//VALVES
// Pump Isolation Valves
// FB_VRC
//EBD Side
//TURBO
fb_AT1K0_GAS_VRC_10(i_xExtILK_OK := F_TurboGateValve_ILK(fb_AT1K0_GAS_PTM_10.iq_stPtm,fb_AT1K0_GAS_GPI_10.PG), i_xOverrideMode := xSystemOverrideMode);
fb_AT1K0_GAS_VRC_20(i_xExtILK_OK := F_TurboGateValve_ILK(fb_AT1K0_GAS_PTM_20.iq_stPtm,fb_AT1K0_GAS_GPI_20.PG), i_xOverrideMode := xSystemOverrideMode);
fb_AT1K0_GAS_VRC_30(i_xExtILK_OK := F_TurboGateValve_ILK(fb_AT1K0_GAS_PTM_30.iq_stPtm,fb_AT1K0_GAS_GPI_30.PG), i_xOverrideMode := xSystemOverrideMode);
fb_AT1K0_GAS_VRC_40(i_xExtILK_OK := F_TurboGateValve_ILK(fb_AT1K0_GAS_PTM_40.iq_stPtm,fb_AT1K0_GAS_GPI_40.PG), i_xOverrideMode := xSystemOverrideMode);
//EBD
fb_AT1K0_GAS_VRC_50(i_xExtILK_OK := F_VRC_DIODE_ILK(fb_AT1K0_GAS_GPI_50.PG,fb_AT1K0_GAS_GPI_51.PG), i_xOverrideMode := xSystemOverrideMode);
fb_AT1K0_GAS_VRC_60(i_xExtILK_OK := F_VRC_DIODE_ILK(fb_AT1K0_GAS_GPI_60.PG,fb_AT1K0_GAS_GPI_51.PG), i_xOverrideMode := xSystemOverrideMode);
//FEE Side
fb_AT1K0_GAS_VRC_70(i_xExtILK_OK := fb_AT1K0_GAS_PMF_90.stPump.i_xMPStatus, i_xOverrideMode := xSystemOverrideMode);
fb_AT1K0_GAS_VRC_90(i_xExtILK_OK := fb_AT1K0_GAS_PMF_90.stPump.i_xMPStatus, i_xOverrideMode := xSystemOverrideMode);
fb_AT1K0_GAS_VRC_100(i_xExtILK_OK := fb_AT1K0_GAS_PMF_100.stPump.i_xMPStatus, i_xOverrideMode := xSystemOverrideMode);
//TURBO
fb_AT1K0_GAS_VRC_110(i_xExtILK_OK := F_TurboGateValve_ILK(fb_AT1K0_GAS_PTM_110.iq_stPtm,fb_AT1K0_GAS_GPI_110.PG), i_xOverrideMode := xSystemOverrideMode);
fb_AT1K0_GAS_VRC_120(i_xExtILK_OK := F_TurboGateValve_ILK(fb_AT1K0_GAS_PTM_120.iq_stPtm,fb_AT1K0_GAS_GPI_120.PG), i_xOverrideMode := xSystemOverrideMode);
fb_AT1K0_GAS_VRC_130(i_xExtILK_OK := F_TurboGateValve_ILK(fb_AT1K0_GAS_PTM_130.iq_stPtm,fb_AT1K0_GAS_GPI_130.PG), i_xOverrideMode := xSystemOverrideMode);
fb_AT1K0_GAS_VRC_140(i_xExtILK_OK := F_TurboGateValve_ILK(fb_AT1K0_GAS_PTM_140.iq_stPtm,fb_AT1K0_GAS_GPI_140.PG) , i_xOverrideMode := xSystemOverrideMode);
//N2 valve
//INL VCN, VGP and VRC_70 are closed.
fb_AT1K0_GAS_VRC_80.i_xExtILK_OK := fb_AT1K0_GAS_VRC_90.iq_stValve.i_xClsLS AND VCN_70.iq_stVCN.rReqPosition <0.4 AND VVC_71.M_IsClosed() AND VVC_72.M_IsClosed() ; //AND VGP is closed;
fb_AT1K0_GAS_VRC_80( i_xOverrideMode := xSystemOverrideMode);


// Turbo Pumps
// FB_PTM_Ebara_010M
//EBD SIDE
fb_AT1K0_GAS_PTM_10(i_xExtILKOk := F_TurboExtILKLogic_2(fb_AT1K0_GAS_PTM_10.iq_stPtm, fb_AT1K0_GAS_GPI_11.PG, fb_AT1K0_GAS_GPI_10.PG,fb_AT1K0_GAS_PMF_10.iq_stPFO));
fb_AT1K0_GAS_PTM_20(i_xExtILKOk := F_TurboExtILKLogic_2(fb_AT1K0_GAS_PTM_20.iq_stPtm, fb_AT1K0_GAS_GPI_11.PG, fb_AT1K0_GAS_GPI_20.PG,fb_AT1K0_GAS_PMF_10.iq_stPFO));
fb_AT1K0_GAS_PTM_30(i_xExtILKOk := F_TurboExtILKLogic_2(fb_AT1K0_GAS_PTM_30.iq_stPtm, fb_AT1K0_GAS_GPI_11.PG, fb_AT1K0_GAS_GPI_30.PG,fb_AT1K0_GAS_PMF_10.iq_stPFO));
fb_AT1K0_GAS_PTM_40(i_xExtILKOk := F_TurboExtILKLogic_2(fb_AT1K0_GAS_PTM_40.iq_stPtm, fb_AT1K0_GAS_GPI_11.PG, fb_AT1K0_GAS_GPI_40.PG,fb_AT1K0_GAS_PMF_10.iq_stPFO));
//FEE Side
fb_AT1K0_GAS_PTM_110(i_xExtILKOk := F_TurboExtILKLogic_2(fb_AT1K0_GAS_PTM_110.iq_stPtm, fb_AT1K0_GAS_GPI_111.PG,fb_AT1K0_GAS_GPI_110.PG,fb_AT1K0_GAS_PMF_110.stPump));
fb_AT1K0_GAS_PTM_120(i_xExtILKOk := F_TurboExtILKLogic_2(fb_AT1K0_GAS_PTM_120.iq_stPtm, fb_AT1K0_GAS_GPI_121.PG, fb_AT1K0_GAS_GPI_120.PG,fb_AT1K0_GAS_PMF_120.stPump));
fb_AT1K0_GAS_PTM_130(i_xExtILKOk := F_TurboExtILKLogic_2(fb_AT1K0_GAS_PTM_130.iq_stPtm, fb_AT1K0_GAS_GPI_121.PG,fb_AT1K0_GAS_GPI_130.PG,fb_AT1K0_GAS_PMF_120.stPump)); 
fb_AT1K0_GAS_PTM_140(i_xExtILKOk := F_TurboExtILKLogic_2(fb_AT1K0_GAS_PTM_140.iq_stPtm, fb_AT1K0_GAS_GPI_141.PG,fb_AT1K0_GAS_GPI_140.PG,fb_AT1K0_GAS_PMF_140.stPump));

// Injector side
fb_AT1K0_GAS_VVC_80(i_xExtILK_OK:= (fb_AT1K0_GAS_PMF_110.stPump.eState = pumpRUNNING  OR  fb_AT1K0_GAS_PMF_110.stPump.eState = pumpSTARTING ) AND (fb_AT1K0_GAS_PTM_80.iq_stPtm.eState = pumpSTARTING OR fb_AT1K0_GAS_PTM_80.iq_stPtm.eState = pumpRUNNING) , i_xOverrideMode:= xSystemOverrideMode , iq_stValve=> );
fb_AT1K0_GAS_PTM_80(i_xExtILKOk := F_TurboExtILKLogic_2(fb_AT1K0_GAS_PTM_80.iq_stPtm, fb_AT1K0_GAS_GPI_111.PG,fb_AT1K0_GAS_GPI_80.PG,fb_AT1K0_GAS_PMF_110.stPump));

//Rouging pumps
// FB_EbaraDryPump
//EBD SIDE
fb_AT1K0_GAS_PMF_10(xExtIlk :=TRUE,TurboIsOn := TRUE);
fb_AT1K0_GAS_PMF_60(xExtIlk :=TRUE,TurboIsOn := TRUE);
//FEE SIDE
fb_AT1K0_GAS_PMF_90(i_stBPGauge := fb_AT1K0_GAS_GPI_90.PG, i_xVlvOpn := TRUE, i_xExtIlkOK := TRUE);
fb_AT1K0_GAS_PMF_100(i_stBPGauge := fb_AT1K0_GAS_GPI_100.PG, i_xVlvOpn := TRUE, i_xExtIlkOK := TRUE);
fb_AT1K0_GAS_PMF_110(i_xExtIlkOK:= TRUE (*Interlock Timer on the Rough Valve*) , stPump=> );
fb_AT1K0_GAS_PMF_120(i_xExtIlkOK:= TRUE(*Interlock Timer on the Rough Valve*), stPump=> );
fb_AT1K0_GAS_PMF_140(i_xExtIlkOK:= TRUE(*Interlock Timer on the Rough Valve*), stPump=> );
if( fb_AT1K0_GAS_PMF_110.stPump.eState = pumpSTARTING ) OR ( fb_AT1K0_GAS_PMF_110.stPump.eState = pumpRUNNING ) THEN fb_AT1K0_GAS_VVC_110.M_Open(TRUE); END_IF
if( fb_AT1K0_GAS_PMF_120.stPump.eState = pumpSTARTING ) OR ( fb_AT1K0_GAS_PMF_120.stPump.eState = pumpRUNNING ) THEN fb_AT1K0_GAS_VVC_120.M_Open(TRUE); END_IF
if( fb_AT1K0_GAS_PMF_140.stPump.eState = pumpSTARTING ) OR ( fb_AT1K0_GAS_PMF_140.stPump.eState = pumpRUNNING ) THEN fb_AT1K0_GAS_VVC_140.M_Open(TRUE); END_IF
fb_AT1K0_GAS_VVC_110(i_xExtILK_OK:= (fb_AT1K0_GAS_PMF_110.stPump.eState = pumpRUNNING  OR  fb_AT1K0_GAS_PMF_110.stPump.eState = pumpSTARTING ), i_xOverrideMode:= , iq_stValve=> );
fb_AT1K0_GAS_VVC_120(i_xExtILK_OK:= (fb_AT1K0_GAS_PMF_120.stPump.eState = pumpRUNNING  OR  fb_AT1K0_GAS_PMF_120.stPump.eState = pumpSTARTING ), i_xOverrideMode:= , iq_stValve=> );
fb_AT1K0_GAS_VVC_140(i_xExtILK_OK:= (fb_AT1K0_GAS_PMF_140.stPump.eState = pumpRUNNING  OR  fb_AT1K0_GAS_PMF_140.stPump.eState = pumpSTARTING ), i_xOverrideMode:= , iq_stValve=> );

END_PROGRAM

// ---- POUs/PRG_INJ.TcPOU
PROGRAM PRG_INJ
VAR
	{attribute 'pytmc' :=' pv: AT1K0:GATT:CNTRL:SP '}
	fSetpointValue :FLOAT; 
	{attribute 'pytmc' :=' pv: AT1K0:GATT:CNTRL:GO;
	 field: ZNAM STOP; 
	 field: ONAM START; 
	 io: io;
	'}
	bGo: BOOL; 
 	{attribute 'pytmc' :=' pv: AT1K0:GATT:CNTRL:RESET;
	 field: ZNAM FALSE; 
	 field: ONAM TRUE; 
	 io: io;
	 '}
	bReset : BOOL; 
	{attribute 'pytmc' :=' pv: AT1K0:GATT:CNTRL:ERROR;
    field: ZNAM FALSE; 
	 field: ONAM TRUE; 
	 io: io;
	 '}
	bError : BOOL; 
	{attribute 'pytmc' :=' pv: AT1K0:GATT:CNTRL:Kp1 '}
	fKp1 : REAL:= 0.04; 
	{attribute 'pytmc' :=' pv: AT1K0:GATT:CNTRL:Tn1 '}
	fTn1 : REAL:= 1;//0.5; 
	{attribute 'pytmc' :=' pv: AT1K0:GATT:CNTRL:Kp2 '}
	fKp2 : REAL:= 0.01; 
	{attribute 'pytmc' :=' pv: AT1K0:GATT:CNTRL:Tn2 '}
	fTn2 : REAL:= 0.5; 
	arrTable	: ARRAY[1..31,1..2] OF FLOAT;
	fManValue											: FLOAT;
	bExtrapolate										: BOOL;
	eMode							: E_CTRL_MODE;
	stCTRL_PID_PARAMS		: ST_CTRL_PID_PARAMS;
	bSync							: BOOL;
	bHold							: BOOL;
	eErrorId						: E_CTRL_ERRORCODES;
	bARWactive					: BOOL;
	(* controller *)
	fbCTRL_PID					: FB_CTRL_PID;
	bInit							: BOOL	:= TRUE;
	fbCTRL_LIN_INTERPOLATION					: FB_CTRL_LIN_INTERPOLATION;
	//stCTRL_LIN_INTERPOLATION_PARAMS		: ST_CTRL_LIN_INTERPOLATION_PARAMS;
	stCTRL_LIN_INTERPOLATION_PARAMS_GEM	: ST_CTRL_LIN_INTERPOLATION_PARAMS;
	fbCTRL_DEADBAND						: FB_CTRL_DEADBAND;
	stCTRL_DEADBAND_PARAMS			: ST_CTRL_DEADBAND_PARAMS;

	pid_on :TON;
	wait : time := T#10S;
	FTrig: F_TRIG;
		

	
END_VAR


// Valves
VCN_70(i_xExtIlkOK := ((US_MAA_OK AND US_Roughing_Valves_Open AND US_Turbo_Valves_Open AND US_Turbo_Running) 
						AND (DS_MAA_OK AND DS_Roughing_Valves_Open AND DS_Turbo_Valves_Open AND DS_Turbo_Running)), 
						i_ReqPos:=  fbCTRL_LIN_INTERPOLATION.fOut + fbCTRL_PID.fOut);

//VGP_80
VVC_71(i_xExtILK_OK:= VVC_72.M_IsClosed(), i_xOverrideMode:= , iq_stValve=> );
VVC_72(i_xExtILK_OK:= VVC_71.M_IsClosed(), i_xOverrideMode:= , iq_stValve=> );

//Gauges
GCM_70(PG=> , i_rFULL_SCALE:= 2000);
GCM_80(PG=> , i_rFULL_SCALE:= 20);
GCM_81(PG=> , i_rFULL_SCALE:= 0.25);
(*Assign reading to psuedo gauge*)
IF (GCM_81.PG.rPRESS >=0.22) THEN GCM_82 := GCM_80.PG;
	ELSE
	GCM_82 := GCM_81.PG;	
END_IF
// Set ADC bits for EL3174-0002
GCM_70.M_SetBits(30518);
GCM_80.M_SetBits(30518);
GCM_81.M_SetBits(30518);


//
(*Iniitialization*)
IF bInit
THEN
	(* init array with the interpolation points  *)
	(* 	fIn					 |		fOut		*)
	arrTable[1,1] := 0;		arrTable[1,2] := 0;
	arrTable[2,1] := 0.0000412;		arrTable[2,2] := 34;
	arrTable[3,1] := 0.001282;		arrTable[3,2] := 36;
	arrTable[4,1] :=  0.002136;	    arrTable[4,2] := 38;
	arrTable[5,1] :=  0.005884;	    arrTable[5,2] := 40;
	arrTable[6,1] := 0.00907;		arrTable[6,2] := 42;
	arrTable[7,1] := 0.01183;		arrTable[7,2] := 44;
	arrTable[8,1] := 0.01799;	    arrTable[8,2] := 46;
	arrTable[9,1] := 0.0302;	    arrTable[9,2] := 47;
	arrTable[10,1] := 0.0417;		arrTable[10,2] := 50;
	arrTable[11,1] := 0.06635;		arrTable[11,2] := 51;
	arrTable[12,1] := 0.08118;		arrTable[12,2] := 53;
	arrTable[13,1] := 0.0998;		arrTable[13,2] := 56;
	arrTable[14,1] := 0.10644;		arrTable[14,2] := 56.5;
	arrTable[15,1] := 0.1359;		arrTable[15,2] := 58;
	arrTable[16,1] := 0.1929;		arrTable[16,2] := 60;
	arrTable[17,1] := 0.2922;		arrTable[17,2] := 62;
	arrTable[18,1] := 0.3428;	    arrTable[18,2] := 64;
	arrTable[19,1] :=  0.405;;	    arrTable[19,2] :=66;
	arrTable[20,1] := 0.481;		arrTable[20,2] := 68;
	arrTable[21,1] := 0.5542;		arrTable[21,2] := 69;
	arrTable[22,1] := 0.6333;	    arrTable[22,2] := 70;
	arrTable[23,1] := 0.7901;	    arrTable[23,2] := 72;
	arrTable[24,1] := 0.9307;		arrTable[24,2] := 73.04;
	arrTable[25,1] := 1.0448;		arrTable[25,2] := 73.64;
	arrTable[26,1] := 1.31919;;		arrTable[26,2] := 74.45;
	arrTable[27,1] :=  1.324;		arrTable[27,2] :=74.46;
	arrTable[28,1] := 1.71941;	arrTable[28,2] := 75;
	arrTable[29,1] :=  1.963194;		arrTable[29,2] :=75.5;
	arrTable[30,1] := 1.99999;	arrTable[30,2] := 75.505;
	arrTable[31,1] := 2;	arrTable[31,2] := 75.55;
	(* init parameter struct *)
	stCTRL_LIN_INTERPOLATION_PARAMS_GEM.tCtrlCycleTime					:= T#10ms;
	stCTRL_LIN_INTERPOLATION_PARAMS_GEM.tTaskCycleTime					:= T#10ms;
	stCTRL_LIN_INTERPOLATION_PARAMS_GEM.nDataTable_NumberOfRows		:= INT_TO_UINT(31);	

	(*FBCNTRL*)
	(* init parameter struct *)
	stCTRL_PID_PARAMS.tCtrlCycleTime		:= T#10ms;
	stCTRL_PID_PARAMS.tTaskCycleTime		:= T#10ms;
	stCTRL_PID_PARAMS.fKp					:= fKp1;			(* proportional gain Kp				*)
	stCTRL_PID_PARAMS.tTn					:= T#500ms;		(*  Tn									*)
	stCTRL_PID_PARAMS.tTv					:= T#200ms;	(*  Tv									*)
	stCTRL_PID_PARAMS.tTd					:= T#100ms;	(*  Td									*)
	stCTRL_PID_PARAMS.fOutMaxLimit			:=  78;			(* maximum output limit				*)
	stCTRL_PID_PARAMS.fOutMinLimit			:=  -100;			(* minimum output limit				*)

	(* set the mode to ACTIVE --> normal operation *)
	eMode							:= eCTRL_MODE_ACTIVE   ;					
	(* reset the init flag *)
	bInit							:= FALSE;
END_IF
(* set the addresses *)
	stCTRL_LIN_INTERPOLATION_PARAMS_GEM.pDataTable_ADR			:= ADR(arrTable);
	stCTRL_LIN_INTERPOLATION_PARAMS_GEM.nDataTable_SIZEOF		:= SIZEOF(arrTable);

if (bGo) THEN
	IF (bReset) THEN
	(* set the mode to RESET*)
	eMode							:= eCTRL_MODE_RESET   ;
	VCN_70.M_ValveControl(CloseValve);
	//bReset := False;
	ELSE
		(* set the mode to ACTIVE --> normal operation *)
	eMode							:= eCTRL_MODE_ACTIVE   ;
 	VCN_70.M_ValveControl(PressureControl);
	END_IF
END_IF
If(FTrig.Q)THEN
		eMode							:= eCTRL_MODE_PASSIVE;
		VCN_70.M_ValveControl(CloseValve);
		fSetpointValue :=0;
END_IF


fbCTRL_LIN_INTERPOLATION(
	fIn:= fSetpointValue , 
	fManValue:= fManValue , 
	bExtrapolate:= bExtrapolate, 
	eMode:= eMode, 
	stParams:= stCTRL_LIN_INTERPOLATION_PARAMS_GEM,
	fOut=> , 
	bInIsGreaterThanMaxElement=> , 
	bInIsLessThanMinElement=> , 
	eState=> , 
	eErrorId=> , 
	bError=> );


(* Gauge selection *)
IF (fSetpointValue >=0.22) THEN
	fbCTRL_PID.fActualValue := GCM_80.PG.rPRESS;
ELSE
	fbCTRL_PID.fActualValue := GCM_81.PG.rPRESS;
END_IF

(* call controller *)
fbCTRL_PID(		fSetpointValue		:= fSetpointValue,
					fActualValue		:= ,
					fManSyncValue	:= ,
					bSync				:= bSync,
					eMode				:= eMode,
					bHold				:= bHold,
					stParams			:= stCTRL_PID_PARAMS,
					fOut				=> ,
					bARWactive		=> bARWactive,
					eErrorId			=> eErrorId,
					bError				=> 
				);

	
(*deadband/clipper *)

(* call function block *)
stCTRL_DEADBAND_PARAMS.fThreshold	:=  fSetpointValue*0.0016 ;
(*fbCTRL_DEADBAND	(	fIn					:= ,
					stParams			:= stCTRL_DEADBAND_PARAMS,
					bInIsUnderThreshold => ,
					eErrorId			=> ,
					bError				=> 
				);*)

bError := fbCTRL_PID.bError OR fbCTRL_LIN_INTERPOLATION.bError;
				

	

// or NOT???

//stCTRL_PID_PARAMS.bDInTheFeedbackPath := fbCTRL_DEADBAND.bInIsUnderThreshold;


//timer
(*pid_on(IN:=, PT:= wait, Q=>, ET =>);
IF (pid_on.Q) THEN eMode:= eCTRL_MODE_ACTIVE; pid_on.IN := FALSE; END_IF; //eCTRL_MODE_TUNE????*)


FTRIG(CLK := bGo);

END_PROGRAM

// ---- POUs/PRG_Motion.TcPOU
PROGRAM PRG_Motion
VAR
	bInit: BOOL := TRUE;
	iReqApperture: INT :=1;
	
	bAllGo : Bool := false;
	
	/////
 (* fbMAX_1: FB_MotionStage;
  fbMAY_1: FB_MotionStage;
  
  fbMAX_2: FB_MotionStage;
  fbMAY_2: FB_MotionStage;
  
  fbMAX_3: FB_MotionStage;
  fbMAY_3: FB_MotionStage;
  
  fbMAX_4: FB_MotionStage;
  fbMAY_4: FB_MotionStage;*)
	
	/////
	{attribute 'pytmc' := '
		pv: MMS:1:STATE
		io: io
	'}
	fbMAA_1_States: FB_MAA;
	{attribute 'pytmc' := '
		pv: MMS:2:STATE
		io: io
	'}
	fbMAA_2_States: FB_MAA;
	{attribute 'pytmc' := '
		pv: MMS:3:STATE
		io: io
	'}
	fbMAA_3_States: FB_MAA;
	{attribute 'pytmc' := '
		pv: MMS:4:STATE
		io: io
	'}
	fbMAA_4_States: FB_MAA;

END_VAR

/// PMPS ???????????
//LIMIT the array index
iReqApperture := LIMIT(1,pv_iReqApperture,4);


(*
IF(bInit) THEN
	// initialise all the values of pre defined positions for each apperture in the assembly array 
	VAA_1_Y_POS[1] :=0;
	VAA_1_Y_POS[2] :=0;
	VAA_1_Y_POS[3] :=0;
	VAA_1_Y_POS[4] :=0;
	
	VAA_2_Y_POS[1] :=0;
	VAA_2_Y_POS[2] :=0;
	VAA_2_Y_POS[3] :=0;
	VAA_2_Y_POS[4] :=0;
	
	VAA_3_Y_POS[1] :=0;
	VAA_3_Y_POS[2] :=0;
	VAA_3_Y_POS[3] :=0;
	VAA_3_Y_POS[4] :=0;
	
	VAA_4_Y_POS[1] :=0;
	VAA_4_Y_POS[2] :=0;
	VAA_4_Y_POS[3] :=0;
	VAA_4_Y_POS[4] :=0;
END_IF


(*No STO*)
M1.bHardwareEnable := TRUE;
M2.bHardwareEnable := TRUE;
M3.bHardwareEnable := TRUE;
M4.bHardwareEnable := TRUE;

M5.bHardwareEnable := TRUE;
M6.bHardwareEnable := TRUE;
M7.bHardwareEnable := TRUE;
M8.bHardwareEnable := TRUE;

(*Instantiate the motion function blocks*)
fbMAX_1(stMotionStage := M1);
fbMAY_1(stMotionStage := M2);

fbMAX_2(stMotionStage := M3);
fbMAY_2(stMotionStage := M4);

fbMAX_3(stMotionStage := M4);
fbMAY_3(stMotionStage := M6);

fbMAX_4(stMotionStage := M7);
fbMAY_4(stMotionStage := M8);

(* PTP to aperture position on the each aperture array assembly*)
fbMAA_1_States(
	stMotionStage:=M2,
	fbGoAprt1:=VAA_1_Y_POS[1],
	fbGoAprt2:=VAA_1_Y_POS[2],
	fbGoAprt3:=VAA_1_Y_POS[3],
	fbGoAprt4:=VAA_1_Y_POS[4]);

fbMAA_2_States(
	stMotionStage:=M4,
	fbGoAprt1:=VAA_2_Y_POS[1],
	fbGoAprt2:=VAA_2_Y_POS[2],
	fbGoAprt3:=VAA_2_Y_POS[3],
	fbGoAprt4:=VAA_2_Y_POS[4]);
	
fbMAA_3_States(
	stMotionStage:=M6,
	fbGoAprt1:=VAA_3_Y_POS[1],
	fbGoAprt2:=VAA_3_Y_POS[2],
	fbGoAprt3:=VAA_3_Y_POS[3],
	fbGoAprt4:=VAA_3_Y_POS[4]);
	
fbMAA_4_States(
	stMotionStage:=M8,
	fbGoAprt1:=VAA_4_Y_POS[1],
	fbGoAprt2:=VAA_4_Y_POS[2],
	fbGoAprt3:=VAA_4_Y_POS[3],
	fbGoAprt4:=VAA_4_Y_POS[4]);
	
If (bAllGo) Then

	CASE iReqApperture of
		
	1:
		fbMAA_1_States.fbGoAprt1.bExecute := TRUE;
		fbMAA_2_States.fbGoAprt1.bExecute := TRUE;
		fbMAA_3_States.fbGoAprt1.bExecute := TRUE;
		fbMAA_4_States.fbGoAprt1.bExecute := TRUE;		
	2:
		fbMAA_1_States.fbGoAprt2.bExecute := TRUE;
		fbMAA_2_States.fbGoAprt2.bExecute := TRUE;
		fbMAA_3_States.fbGoAprt2.bExecute := TRUE;
		fbMAA_4_States.fbGoAprt2.bExecute := TRUE;	
	
	3:
		fbMAA_1_States.fbGoAprt3.bExecute := TRUE;
		fbMAA_2_States.fbGoAprt3.bExecute := TRUE;
		fbMAA_3_States.fbGoAprt3.bExecute := TRUE;
		fbMAA_4_States.fbGoAprt3.bExecute := TRUE;	
	
	4:
		fbMAA_1_States.fbGoAprt4.bExecute := TRUE;
		fbMAA_2_States.fbGoAprt4.bExecute := TRUE;
		fbMAA_3_States.fbGoAprt4.bExecute := TRUE;
		fbMAA_4_States.fbGoAprt4.bExecute := TRUE;	
	
	END_CASE

END_IF
*)

END_PROGRAM

// ---- POUs/PRG_ILK.TcPOU
PROGRAM PRG_ILK
VAR
END_VAR

(*Evaluate Global Interlocks*)

//TwinscrewPumps_Valves_Closed := GEM1_VRC_60.q_stValve.i_xClsLS AND  GEM1_VRC_70.q_stValve.i_xClsLS AND GEM2_VRC_10.q_stValve.i_xClsLS AND GEM2_VRC_20.q_stValve.i_xClsLS;
US_MAA_OK := TRUE;
DS_MAA_OK := TRUE ;
US_Roughing_Valves_Open := (fb_AT1K0_GAS_VRC_50.i_xOpnLS AND fb_AT1K0_GAS_VRC_60.i_xOpnLS);
DS_Roughing_Valves_Open := (fb_AT1K0_GAS_VRC_90.iq_stValve.i_xOpnLS AND( fb_AT1K0_GAS_PMF_90.stPump.eState := pumpRUNNING)) OR   (fb_AT1K0_GAS_VRC_100.iq_stValve.i_xOpnLS AND (fb_AT1K0_GAS_PMF_100.stPump.eState := pumpRUNNING ));
US_Turbo_Valves_Open := fb_AT1K0_GAS_VRC_10.iq_stValve.i_xOpnLS AND  fb_AT1K0_GAS_VRC_20.iq_stValve.i_xOpnLS AND fb_AT1K0_GAS_VRC_30.iq_stValve.i_xOpnLS AND fb_AT1K0_GAS_VRC_40.iq_stValve.i_xOpnLS;
DS_Turbo_Valves_Open := fb_AT1K0_GAS_VRC_110.iq_stValve.i_xOpnLS AND  fb_AT1K0_GAS_VRC_120.iq_stValve.i_xOpnLS AND fb_AT1K0_GAS_VRC_130.iq_stValve.i_xOpnLS AND fb_AT1K0_GAS_VRC_140.iq_stValve.i_xOpnLS; 
US_Turbo_Running := (fb_AT1K0_GAS_PTM_10.iq_stPtm.eState = pumpRUNNING) AND (fb_AT1K0_GAS_PTM_20.iq_stPtm.eState = pumpRUNNING) AND (fb_AT1K0_GAS_PTM_30.iq_stPtm.eState = pumpRUNNING) AND (fb_AT1K0_GAS_PTM_40.iq_stPtm.eState = pumpRUNNING);
DS_Turbo_Running := (fb_AT1K0_GAS_PTM_110.iq_stPtm.eState = pumpRUNNING) AND (fb_AT1K0_GAS_PTM_120.iq_stPtm.eState = pumpRUNNING) AND (fb_AT1K0_GAS_PTM_130.iq_stPtm.eState = pumpRUNNING) AND (fb_AT1K0_GAS_PTM_140.iq_stPtm.eState = pumpRUNNING); (*MG 03.09.20 Turbo is failing, but injection can run without it*)

//xGEM1_AperturesOpnOK := NOT GEM1_VVC_40.iq_stValve.q_xOPN_DO AND NOT GATT_VVC_10.iq_stValve.q_xOPN_DO; //AND VCN is closed 
//xGEM2_AperturesOpnOK := NOT GEM2_VVC_40.iq_stValve.q_xOPN_DO AND NOT GATT_VVC_10.iq_stValve.q_xOPN_DO; //AND VCN is closed 

(* Link The correct override bit to the correct vacuum section*)



(*P/MPS FF*)

END_PROGRAM

// ---- POUs/Test/FB_ILK_TEST.TcPOU
FUNCTION_BLOCK FB_ILK_TEST
VAR_INPUT
END_VAR
VAR_OUTPUT
END_VAR
VAR
END_VAR

END_FUNCTION_BLOCK
